Fanuc KAREL source: port_LDI.kl

PROGRAM TP
%NOLOCKGROUP
VAR
 x: BOOLEAN
BEGIN
 x = LDI[3]
END TP
